// TIA Portal V17 export
// export: Created 2023-06-23T18:33:42.7079367Z, ExportSetting WithDefaults, DisplayName Totally Integrated Automation Portal, DisplayVersion V17, DisplayName TIA Portal Openness, DisplayVersion V17, DisplayName TIA Portal Version Control Interface, DisplayVersion V17, DisplayName STEP 7 Professional, DisplayVersion V17, DisplayName STEP 7 Safety, DisplayVersion V17, DisplayName WinCC Advanced / Unified PC, DisplayVersion V17
VAR_GLOBAL   // PLC tag table "Level"
   iSP1 AT %I16.3 : Bool;
   iSP2 AT %I16.4 : Bool;
   iSA1 AT %I16.5 : Bool;
   iSA2 AT %I16.6 : Bool;
   iSA3 AT %I16.7 : Bool;
   iTM1a AT %I17.0 : Bool;
   iTM1b AT %I17.1 : Bool;
END_VAR
